INTERFACE I_Mc2SlaveAxis EXTENDS I_Mc2Axis_PTP, I_Mc2AxisGear

END_INTERFACE

(* stored: Version 1.1.0.1, ProductVersion 3.1.4026.20
   Itf I_Mc2SlaveAxis: Id {ab3b7ac8-6915-4490-8138-9b7b87406399} *)
